PROGRAM MAIN
VAR
	PDxx : FB_PDxx:= (stCANopenDevice := (AmsNetId:='10.3.0.21.2.1', PortNr := 16#1001));
		
END_VAR


PDxx();

END_PROGRAM

(* stored: Version 1.1.0.1, ProductVersion 3.1.4024.12
   POU MAIN: Id {a29f7abe-562f-42e7-8426-b06f74325e38}, SpecialFunc None *)
